// TIA Portal V18 export
// export: Created 2026-06-22T15:41:34.3020206Z, ExportSetting WithDefaults, DisplayName Totally Integrated Automation Portal, DisplayVersion V18, DisplayName TIA Portal Openness, DisplayVersion V18, DisplayName TIA Portal Version Control Interface, DisplayVersion V18, DisplayName STEP 7 Professional, DisplayVersion V18, DisplayName STEP 7 Safety, DisplayVersion V18, DisplayName WinCC Professional, DisplayVersion V18
VAR_GLOBAL   // PLC tag table "PLC1_Tags"
   Start_Cmd AT %M0.0 : Bool;
   Stop_Cmd AT %M0.1 : Bool;
   bMotorRunning AT %M0.2 : Bool;
   Reset_Cmd AT %M0.3 : Bool;
   DIR_Cmd AT %M0.4 : Bool;
   PID_Setpoint AT %MD10 : Real;
   PID_ProcessValue AT %MD14 : Real;
   PID_Output AT %MD18 : Real;
   Speed_SP_toSend AT %MD22 : Real;
   Speed_PV_from2 AT %MD26 : Real;
   ATV12_Status AT %MW30 : Word;
   Control_Byte AT %MB32 : Byte;
   Clock_1Hz AT %M100.5 : Bool;
   GET_NDR AT %M1.0 : Bool;
   GET_Error AT %M1.1 : Bool;
   GET_Status AT %MW2 : Word;
   PUT_NDR AT %M1.2 : Bool;
   PUT_Error AT %M1.3 : Bool;
   PUT_Status AT %MW4 : Word;
END_VAR
